(* PLC project v0.6.04_CycleSemiAuto.project, CODESYS CODESYS V3.5 SP19 Patch 1 *)
(* stored: creationDateTime 2026-08-11T18:19:14.772569, modificationDateTime 2026-08-11T18:19:14.772569 *)

(* ═══════════════════════════════════════════════════════════════ 🔁 FB_Filter_PT1 — Filtre passe-bas premier ordre (PT1 numérique) ─────────────────────────────────────────────────────────────── 📄 Extrait depuis le projet CODESYS (Device.export, JOYSTICK/) 🎯 Filtre exponentiel discret : y[k] = α·x[k] + (1-α)·y[k-1] où α = CycleTimeS / (T + CycleTimeS), T = TimeConst en secondes. ⚠️ Si TimeConst = 0 ou CycleTimeS = 0, sortie = entrée (pass-through). ═══════════════════════════════════════════════════════════════ 📄 Docs : DOC/AF/AF_Partie-08_Fonction_Joystick_v2.0.md *)
FUNCTION_BLOCK FB_Filter_PT1
  VAR_INPUT
    ValueIn : REAL;  (* / Consigne brute entrée *)
    TimeConst : TIME;  (* / Constante de temps du filtre *)
    CycleTimeS : REAL;  (* / Temps de cycle réel en secondes *)
  END_VAR
  VAR_OUTPUT
    ValueOut : REAL;  (* / Consigne filtrée sortie *)
  END_VAR
  VAR
    T : REAL;
    Alpha : REAL;
  END_VAR

            

T := TIME_TO_REAL(TimeConst) / 1000.0; // ms → s

IF T <= 0.0 OR CycleTimeS <= 0.0 THEN
    ValueOut := ValueIn;
ELSE
    Alpha    := CycleTimeS / (T + CycleTimeS);
    ValueOut := Alpha * ValueIn + (1.0 - Alpha) * ValueOut;
END_IF;

          
END_FUNCTION_BLOCK
